// TIA Portal V17 export
// export: Created 2022-07-28T18:03:17.5467696Z, ExportSetting None, DisplayName Totally Integrated Automation Portal, DisplayVersion V17, DisplayName TIA Portal Openness, DisplayVersion V17, DisplayName TIA Portal Teamcenter Gateway, DisplayVersion V17, DisplayName TIA Portal Version Control Interface, DisplayVersion V17, DisplayName TIA Portal Test Suite Advanced, DisplayVersion V17, DisplayName SINAMICS Startdrive Advanced, DisplayVersion V17, DisplayName SINAMICS DCC, DisplayVersion V17, DisplayName SINAMICS Startdrive G130, G150, S120, S150, SINAMICS MV, S210, DisplayVersion V17, DisplayName SINAMICS Startdrive G110M, G120, G120C, G120D, G120P, G115D, DisplayVersion V17, DisplayName STEP 7 Professional, DisplayVersion V17, DisplayName SIMATIC Energy Suite, DisplayVersion V17, DisplayName STEP 7 CFC, DisplayVersion V17, DisplayName STEP 7 Safety, DisplayVersion V17, DisplayName WinCC Advanced / Unified PC, DisplayVersion V17, DisplayName SIMATIC Visualization Architect, DisplayVersion V17
TYPE "Lib_PLC_CycleInfo"
   STRUCT
      CMD_GLOBAL { ExternalAccessible := 'False'; ExternalVisible := 'False'; ExternalWritable := 'False'} : Int;   // Для Obj - встановлюється на початку циклу із CMD_GLOBAL_SP
      CMD_GLOBAL_SP : Int;   // Комадни у правління із верхнього рівня (управляння групою, ....)
      STW { ExternalWritable := 'False'} : DWord;
      State { ExternalAccessible := 'False'; ExternalVisible := 'False'; ExternalWritable := 'False'} : "Lib_PLC_State";
      Alarm { ExternalAccessible := 'False'; ExternalVisible := 'False'; ExternalWritable := 'False'} : "Lib_PLC_Alarm";   // біти алармів
      "Counter" { ExternalWritable := 'False'} : "Lib_PLC_AlarmCounter";
   END_STRUCT;
END_TYPE
